FUNCTION_BLOCK CS3_Multicast (* Composite Function Block Type *)
  (* Standard: 61499-2 *)
  (* Version 0.2, 2003-12-05, JHC, Rockwell Automation, Renamed from NEWCOMPFB. *)
  (* Version 0.1, 2002-01-08, JHC, Rockwell Automation, Added DLY FB as example. *)
  (* Version 0.0, 2000-05-27, JHC, Rockwell Automation *)
  (* Compiler header: package fb.rt.cs725; *)
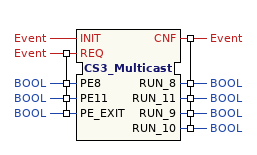
  EVENT_INPUT
    INIT; (* Initialization Request *)
    REQ WITH PE8, PE11, PE_EXIT; (* Normal Execution Request *)
  END_EVENT
  EVENT_OUTPUT
    CNF WITH RUN_8, RUN_11, RUN_9, RUN_10; (* Execution Confirmation *)
  END_EVENT
  VAR_INPUT
    PE8 : BOOL;
    PE11 : BOOL;
    PE_EXIT : BOOL;
  END_VAR
  VAR_OUTPUT
    RUN_8 : BOOL;
    RUN_11 : BOOL;
    RUN_9 : BOOL;
    RUN_10 : BOOL;
  END_VAR
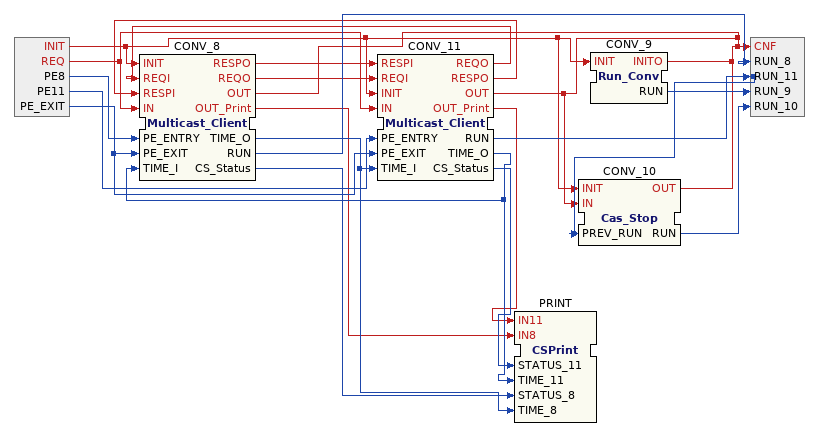
  FBS
    CONV_8 : Multicast_Client;
    CONV_11 : Multicast_Client;
    CONV_9 : Run_Conv;
    CONV_10 : Cas_Stop;
    PRINT : CSPrint;
  END_FBS
  EVENT_CONNECTIONS
    CONV_8.RESPO TO CONV_11.RESPI;
    CONV_8.REQO TO CONV_11.REQI;
    INIT TO CONV_8.INIT;
    INIT TO CONV_11.INIT;
    CONV_11.REQO TO CONV_8.REQI;
    CONV_11.RESPO TO CONV_8.RESPI;
    REQ TO CONV_8.IN;
    CONV_8.OUT TO CNF;
    CONV_11.OUT TO CNF;
    REQ TO CONV_11.IN;
    INIT TO CONV_9.INIT;
    CONV_9.INITO TO CNF;
    INIT TO CONV_10.INIT;
    CONV_10.OUT TO CNF;
    CONV_11.OUT TO CONV_10.IN;
    CONV_11.OUT_Print TO PRINT.IN11;
    CONV_8.OUT_Print TO PRINT.IN8;
  END_CONNECTIONS
  DATA_CONNECTIONS
    PE8 TO CONV_8.PE_ENTRY;
    PE_EXIT TO CONV_8.PE_EXIT;
    PE11 TO CONV_11.PE_ENTRY;
    PE_EXIT TO CONV_11.PE_EXIT;
    CONV_11.RUN TO RUN_11;
    CONV_11.TIME_O TO CONV_8.TIME_I;
    CONV_8.TIME_O TO CONV_11.TIME_I;
    CONV_8.RUN TO RUN_8;
    CONV_9.RUN TO RUN_9;
    RUN_11 TO CONV_10.PREV_RUN;
    CONV_10.RUN TO RUN_10;
    CONV_11.CS_Status TO PRINT.STATUS_11;
    CONV_11.TIME_O TO PRINT.TIME_11;
    CONV_8.CS_Status TO PRINT.STATUS_8;
    CONV_8.TIME_O TO PRINT.TIME_8;
  END_CONNECTIONS
END_FUNCTION_BLOCK
